TYPE "PositioningMachine_Wng"
VERSION : 0.1
// Block: PositioningMachine_Wng
   STRUCT
      NotAutReady : Bool;
      AxisNotInOperation : Bool;
      MissingCnd_BWD : Bool;
      MissingCnd_FWD : Bool;
      Ax : TAx_Warnings;
   END_STRUCT;

END_TYPE
